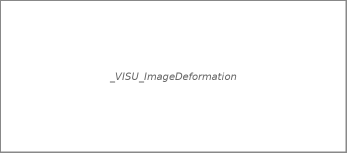
VISUALIZATION _VISU_ContainerDefGrid  // 347x153
VAR_IN_OUT
	m_Inst : FB_ContainerDefGrid;
END_VAR
    Frame (0,0 347x153)
        shows _VISU_ImageDeformation(m_Inst := m_Inst.fBImageDeformation)
END_VISUALIZATION

(* stored: Version 1.1.0.1, ProductVersion 3.1.4024.3
   Visu _VISU_ContainerDefGrid: Id {c50a27c5-b858-44a4-a87d-9622002e5bd8} *)
